FUNCTION_BLOCK _ETcVn2dCodeSearchStrategy_TestSuite EXTENDS TcUnit.FB_TestSuite
VAR
END_VAR

TestAddress();
TestClearReference();
TestClone();
TestTypeNameReturnsExpected();
TestIdentifierReturnsExpected();
TestMakeReferenceToFollowsReference();
TestMakeReferenceToUpdatesReference();
TestSize();
TestValueReturnsExpectedAfterInit();
TestValueReturnsExpectedAfterChange();
TestSerializeTypeWith();
TestSerializeWith();
TestTryDeserializeFrom();
TestTryMakeReferenceToFollowsReference();
TestTryMakeReferenceToUpdatesReference();

METHOD PUBLIC TestAddress
VAR
    _type : _ETcVn2dCodeSearchStrategy(ETcVn2dCodeSearchStrategy.TCVN_CSS_DEFAULT);
    notExpected : PVOID := 0;
    actual : PVOID;
END_VAR
TEST('TestAddress');

actual := _type.Address;

AssertFalse(
    Condition := (notExpected = actual),
    Message := 'Type did not return a valid address.'
);

TEST_FINISHED();
END_METHOD

METHOD PUBLIC TestClearReference
VAR
    _type : _ETcVn2dCodeSearchStrategy(ETcVn2dCodeSearchStrategy.TCVN_CSS_DEFAULT);
	target : ETcVn2dCodeSearchStrategy := ETcVn2dCodeSearchStrategy.TCVN_CSS_DEFAULT;
    expected : ETcVn2dCodeSearchStrategy := ETcVn2dCodeSearchStrategy.TCVN_CSS_DEFAULT;
    actual : ETcVn2dCodeSearchStrategy;
END_VAR
TEST('TestClearReference');

_type.MakeReferenceTo(target);
_type.ClearReference();
target := ETcVn2dCodeSearchStrategy.TCVN_CSS_FIRST_FLIPPED;

actual := _type.Value;

AssertEquals(
    Expected := expected,
    Actual := actual,
    Message := 'Value continued to follow target.'
);

TEST_FINISHED();
END_METHOD

METHOD PUBLIC TestClone
VAR
    _type : _ETcVn2dCodeSearchStrategy(ETcVn2dCodeSearchStrategy.TCVN_CSS_DEFAULT);
	clone : I_Datatype;
	isValidClone : BOOL;
	compareResult : DINT;
END_VAR
TEST('TestClone');

clone := _type.Clone();

isValidClone := clone <> 0;

IF isValidClone THEN
	compareResult := memcmp(_type.Address, clone.Address, clone.Size);
END_IF

AssertTrue(
	Condition := isValidClone,
	Message := 'Clone did not produce a clone'
);

AssertEquals_DINT(
	Expected := 0,
    Actual := compareResult,
    Message := 'Clone did not return a valid clone.'
);

clone.Dispose();

TEST_FINISHED();
END_METHOD

METHOD PUBLIC TestIdentifierReturnsExpected
VAR
    _type : _ETcVn2dCodeSearchStrategy(ETcVn2dCodeSearchStrategy.TCVN_CSS_DEFAULT);
    expected : STRING := 'ETcVn2dCodeSearchStrategy';
    actual : STRING;
END_VAR
TEST('TestIdentifierReturnsExpected');

actual := _type.Identifier;

AssertEquals_STRING(
    Expected := expected,
    Actual := actual,
    Message := 'Type did not return correct iec type.'
);

TEST_FINISHED();
END_METHOD

METHOD PUBLIC TestMakeReferenceToFollowsReference
VAR
    _type : _ETcVn2dCodeSearchStrategy(ETcVn2dCodeSearchStrategy.TCVN_CSS_DEFAULT);
	target : ETcVn2dCodeSearchStrategy := ETcVn2dCodeSearchStrategy.TCVN_CSS_DEFAULT;
    expected : ETcVn2dCodeSearchStrategy := ETcVn2dCodeSearchStrategy.TCVN_CSS_FIRST_FLIPPED;
    actual : ETcVn2dCodeSearchStrategy;
END_VAR
TEST('TestMakeReferenceToFollowsReference');

_type.MakeReferenceTo(target);
target := ETcVn2dCodeSearchStrategy.TCVN_CSS_FIRST_FLIPPED;

actual := _type.Value;

AssertEquals(
    Expected := expected,
    Actual := actual,
    Message := 'Value did not follow target change.'
);

TEST_FINISHED();
END_METHOD

METHOD PUBLIC TestMakeReferenceToUpdatesReference
VAR
    _type : _ETcVn2dCodeSearchStrategy(ETcVn2dCodeSearchStrategy.TCVN_CSS_DEFAULT);
	target : ETcVn2dCodeSearchStrategy := ETcVn2dCodeSearchStrategy.TCVN_CSS_DEFAULT;
    expected : ETcVn2dCodeSearchStrategy := ETcVn2dCodeSearchStrategy.TCVN_CSS_FIRST_FLIPPED;
    actual : ETcVn2dCodeSearchStrategy;
END_VAR
TEST('TestMakeReferenceToUpdatesReference');

_type.MakeReferenceTo(target);
_type.Value := ETcVn2dCodeSearchStrategy.TCVN_CSS_FIRST_FLIPPED;

actual := target;

AssertEquals(
    Expected := expected,
    Actual := actual,
    Message := 'Value did not update target.'
);

TEST_FINISHED();
END_METHOD

METHOD PUBLIC TestSerializeTypeWith
VAR
    _type : _ETcVn2dCodeSearchStrategy(ETcVn2dCodeSearchStrategy.TCVN_CSS_DEFAULT);
    serializer : JsonSerializer;
    expected : STRING(500) := '{"typeName":"ENUM","identifier":"ETcVn2dCodeSearchStrategy","enumerations":["TCVN_CSS_DEFAULT","TCVN_CSS_FIRST_FLIPPED","TCVN_CSS_FIRST_INVERTED","TCVN_CSS_FIRST_NOT_FLIPPED","TCVN_CSS_FIRST_NOT_INVERTED","TCVN_CSS_ONLY_FLIPPED","TCVN_CSS_ONLY_INVERTED","TCVN_CSS_ONLY_NOT_FLIPPED","TCVN_CSS_ONLY_NOT_INVERTED"],"baseType":{"typeName":"UDINT","minValue":0,"maxValue":4294967295,"isSigned":false,"isFloat":false}}';
    actual : STRING(500);
END_VAR
TEST('TestSerializeTypeWith');

serializer.Reset();
_type.SerializeTypeWith(serializer);
serializer.TryGetSerializedData(ADR(actual), SIZEOF(actual));

AssertEquals_STRING(
    Expected := expected,
    Actual := actual,
    Message := 'Serialization of type did not return correct string.'
);

TEST_FINISHED();
END_METHOD

METHOD PUBLIC TestSerializeWith
VAR
    _type : _ETcVn2dCodeSearchStrategy(ETcVn2dCodeSearchStrategy.TCVN_CSS_DEFAULT);
    serializer : JsonSerializer;
    expected : STRING := '"TCVN_CSS_DEFAULT"';
    actual : STRING(500);
END_VAR
TEST('TestSerializeWith');

serializer.Reset();
_type.SerializeWith(serializer);
serializer.TryGetSerializedData(ADR(actual), SIZEOF(actual));

AssertEquals_STRING(
    Expected := expected,
    Actual := actual,
    Message := 'Serialization of type data did not return correct string.'
);

TEST_FINISHED();
END_METHOD

METHOD PUBLIC TestSize
VAR
    _type : _ETcVn2dCodeSearchStrategy(ETcVn2dCodeSearchStrategy.TCVN_CSS_DEFAULT);
    expected : UDINT := SIZEOF(ETcVn2dCodeSearchStrategy);
    actual : UDINT;
END_VAR
TEST('TestSize');

actual := _type.Size;

AssertEquals_UDINT(
    Expected := Expected,
    Actual := actual,
    Message := 'Type did not return the correct size.'
);

TEST_FINISHED();
END_METHOD

METHOD PUBLIC TestTryDeserializeFrom
VAR
    deserializer : JsonDeserializer;
    feedback : DeserializerFeedback;
    json : STRING := '"TCVN_CSS_DEFAULT"';
    _type : _ETcVn2dCodeSearchStrategy(ETcVn2dCodeSearchStrategy.TCVN_CSS_DEFAULT);
    expected : ETcVn2dCodeSearchStrategy := ETcVn2dCodeSearchStrategy.TCVN_CSS_DEFAULT;
    actual : ETcVn2dCodeSearchStrategy;
 END_VAR
TEST('TestTryDeserializeFrom');

deserializer.Reset();
deserializer.TryLoad(json);
_type.TryDeserializeFrom(Deserializer, Feedback);

actual := _type.Value;

AssertEquals(
    Expected := expected,
    Actual := actual,
    Message := 'Type did not deserialize correctly.'
);

TEST_FINISHED();
END_METHOD

METHOD PUBLIC TestTryMakeReferenceToFollowsReference
VAR
    _type : _ETcVn2dCodeSearchStrategy(ETcVn2dCodeSearchStrategy.TCVN_CSS_DEFAULT);
	target : _ETcVn2dCodeSearchStrategy(ETcVn2dCodeSearchStrategy.TCVN_CSS_DEFAULT);
    expected : ETcVn2dCodeSearchStrategy := ETcVn2dCodeSearchStrategy.TCVN_CSS_FIRST_FLIPPED;
    actual : ETcVn2dCodeSearchStrategy;
END_VAR
TEST('TestTryMakeReferenceToFollowsReference');

_type.TryMakeReferenceTo(target);
target.Value := ETcVn2dCodeSearchStrategy.TCVN_CSS_FIRST_FLIPPED;

actual := _type.Value;

AssertEquals(
    Expected := expected,
    Actual := actual,
    Message := 'Value did not follow target change.'
);

TEST_FINISHED();
END_METHOD

METHOD PUBLIC TestTryMakeReferenceToUpdatesReference
VAR
    _type : _ETcVn2dCodeSearchStrategy(ETcVn2dCodeSearchStrategy.TCVN_CSS_DEFAULT);
	target : _ETcVn2dCodeSearchStrategy(ETcVn2dCodeSearchStrategy.TCVN_CSS_DEFAULT);
    expected : ETcVn2dCodeSearchStrategy := ETcVn2dCodeSearchStrategy.TCVN_CSS_FIRST_FLIPPED;
    actual : ETcVn2dCodeSearchStrategy;
END_VAR
TEST('TestTryMakeReferenceToUpdatesReference');

_type.TryMakeReferenceTo(target);
_type.Value := ETcVn2dCodeSearchStrategy.TCVN_CSS_FIRST_FLIPPED;

actual := target.Value;

AssertEquals(
    Expected := expected,
    Actual := actual,
    Message := 'Value did not update target.'
);

TEST_FINISHED();
END_METHOD

METHOD PUBLIC TestTypeNameReturnsExpected
VAR
    _type : _ETcVn2dCodeSearchStrategy(ETcVn2dCodeSearchStrategy.TCVN_CSS_DEFAULT);
    expected : STRING := 'ENUM';
    actual : STRING;
END_VAR
TEST('TestTypeNameReturnsExpected');

actual := _type.TypeName;

AssertEquals_STRING(
    Expected := expected,
    Actual := actual,
    Message := 'Type did not return correct iec type.'
);

TEST_FINISHED();
END_METHOD

METHOD PUBLIC TestValueReturnsExpectedAfterChange
VAR
    _type : _ETcVn2dCodeSearchStrategy(ETcVn2dCodeSearchStrategy.TCVN_CSS_DEFAULT);
    expected : ETcVn2dCodeSearchStrategy := ETcVn2dCodeSearchStrategy.TCVN_CSS_FIRST_FLIPPED;
    actual : ETcVn2dCodeSearchStrategy;
END_VAR
TEST('TestValueReturnsExpectedAfterChange');

_type.Value := ETcVn2dCodeSearchStrategy.TCVN_CSS_FIRST_FLIPPED;

actual := _type.Value;

AssertEquals(
    Expected := expected,
    Actual := actual,
    Message := 'Expected value not returned after change.'
);

TEST_FINISHED();
END_METHOD

METHOD PUBLIC TestValueReturnsExpectedAfterInit
VAR
    _type : _ETcVn2dCodeSearchStrategy(ETcVn2dCodeSearchStrategy.TCVN_CSS_DEFAULT);
    expected : ETcVn2dCodeSearchStrategy := ETcVn2dCodeSearchStrategy.TCVN_CSS_DEFAULT;
    actual : ETcVn2dCodeSearchStrategy;
END_VAR
TEST('TestValueReturnsExpectedAfterInit');

actual := _type.Value;

AssertEquals(
    Expected := expected,
    Actual := actual,
    Message := 'Expected value not returned after Init.'
);

TEST_FINISHED();
END_METHOD

END_FUNCTION_BLOCK

(* stored: Version 1.1.0.1, ProductVersion 3.1.4024.12
   POU _ETcVn2dCodeSearchStrategy_TestSuite: Id {3d13e6dd-7ed8-4683-b29d-58820479502c}, SpecialFunc None
   Method TestAddress: Id {bcf16a83-c8b2-4cc3-bde9-52d6f6407341}
   Method TestClearReference: Id {95905ee2-41c3-49bd-850c-bc0ccd88c41b}
   Method TestClone: Id {ae5cfe81-edbc-4800-860f-0b5bccd55df0}
   Method TestIdentifierReturnsExpected: Id {f8cb0742-5ba6-4958-81d3-ae11a68f6459}
   Method TestMakeReferenceToFollowsReference: Id {5f74d4dc-4fed-4900-95d3-35fcefea26e6}
   Method TestMakeReferenceToUpdatesReference: Id {92ec4c0e-d8ba-4e06-a665-96d419628935}
   Method TestSerializeTypeWith: Id {3474c79d-9e5d-45b8-b57c-7b389353e7e9}
   Method TestSerializeWith: Id {5d00f0db-50b6-48e2-871b-78e9866f86f6}
   Method TestSize: Id {38ef7745-db12-4e54-aed5-ebd4232883ff}
   Method TestTryDeserializeFrom: Id {b97d1655-2709-4cdf-8d90-093054877d6e}
   Method TestTryMakeReferenceToFollowsReference: Id {b6389b7a-80be-464d-87bf-bdd23a92e080}
   Method TestTryMakeReferenceToUpdatesReference: Id {7ed879be-e5be-4d7f-95d6-18ff75235ba0}
   Method TestTypeNameReturnsExpected: Id {6b10e75e-6ced-446b-9a48-3043e04559ed}
   Method TestValueReturnsExpectedAfterChange: Id {026ee19f-6ba1-40ec-9a75-4988486154d0}
   Method TestValueReturnsExpectedAfterInit: Id {1b4226f3-dedc-4287-869b-ffa5c199543f} *)
